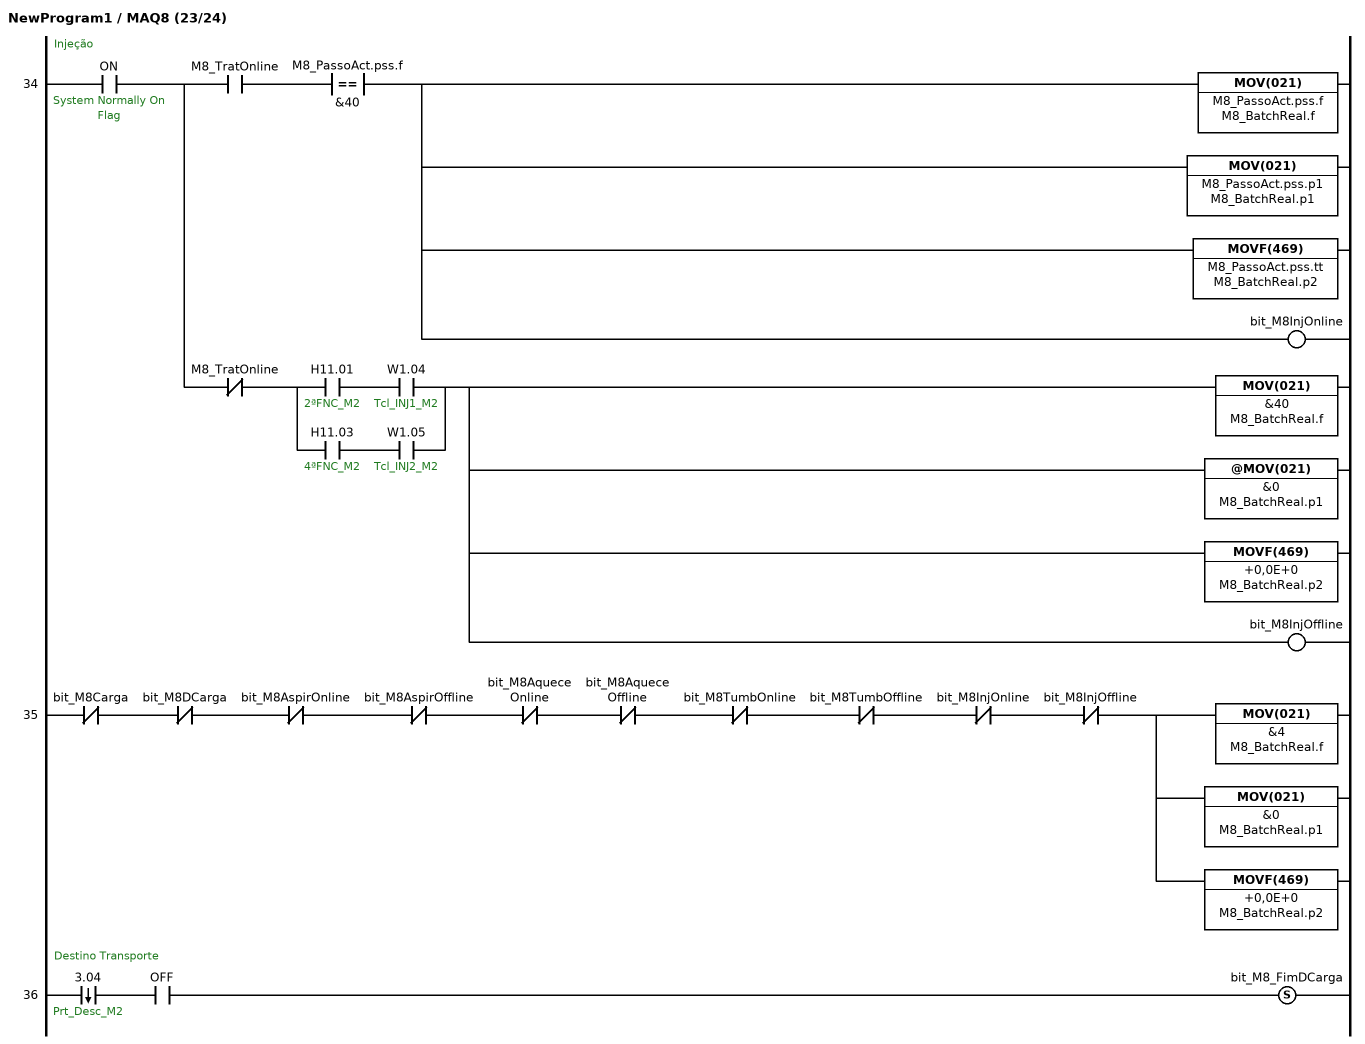
; [picture p48: NewProgram1 / MAQ8, rungs 34-36]
; rung 34: Injeção
LD ON  ; System Normally On Flag
OUT TR0
AND M8_TratOnline
AND=(300) M8_PassoAct.pss.f &40
MOV(021) M8_PassoAct.pss.f M8_BatchReal.f
MOV(021) M8_PassoAct.pss.p1 M8_BatchReal.p1
MOVF(469) M8_PassoAct.pss.tt M8_BatchReal.p2
OUT bit_M8InjOnline
LD TR0
ANDNOT M8_TratOnline
LD H11.01  ; 2ªFNC_M2
AND W1.04  ; Tcl_INJ1_M2
LD H11.03  ; 4ªFNC_M2
AND W1.05  ; Tcl_INJ2_M2
ORLD
ANDLD
MOV(021) &40 M8_BatchReal.f
@MOV(021) &0 M8_BatchReal.p1
MOVF(469) +0,0E+0 M8_BatchReal.p2
OUT bit_M8InjOffline
; rung 35
LDNOT bit_M8Carga
ANDNOT bit_M8DCarga
ANDNOT bit_M8AspirOnline
ANDNOT bit_M8AspirOffline
ANDNOT bit_M8AqueceOnline
ANDNOT bit_M8AqueceOffline
ANDNOT bit_M8TumbOnline
ANDNOT bit_M8TumbOffline
ANDNOT bit_M8InjOnline
ANDNOT bit_M8InjOffline
MOV(021) &4 M8_BatchReal.f
MOV(021) &0 M8_BatchReal.p1
MOVF(469) +0,0E+0 M8_BatchReal.p2
; rung 36: Destino Transporte
%LD 3.04  ; Prt_Desc_M2
AND OFF
SET bit_M8_FimDCarga

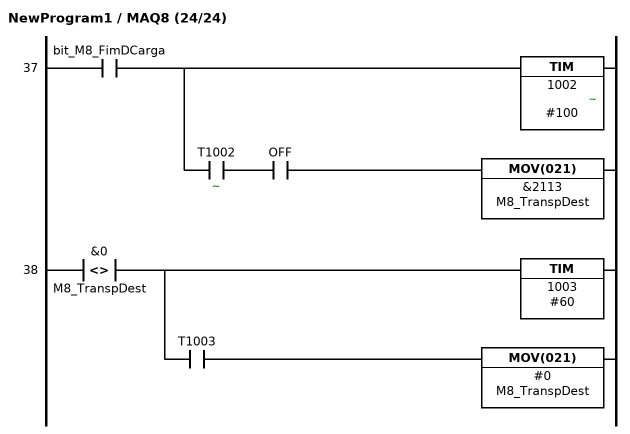
; rung 37
LD bit_M8_FimDCarga
TIM 1002 #100  ; ~
AND T1002  ; ~
AND OFF
MOV(021) &2113 M8_TranspDest
; rung 38
LD<>(305) &0 M8_TranspDest
TIM 1003 #60
AND T1003
MOV(021) #0 M8_TranspDest

### Section TAPETES

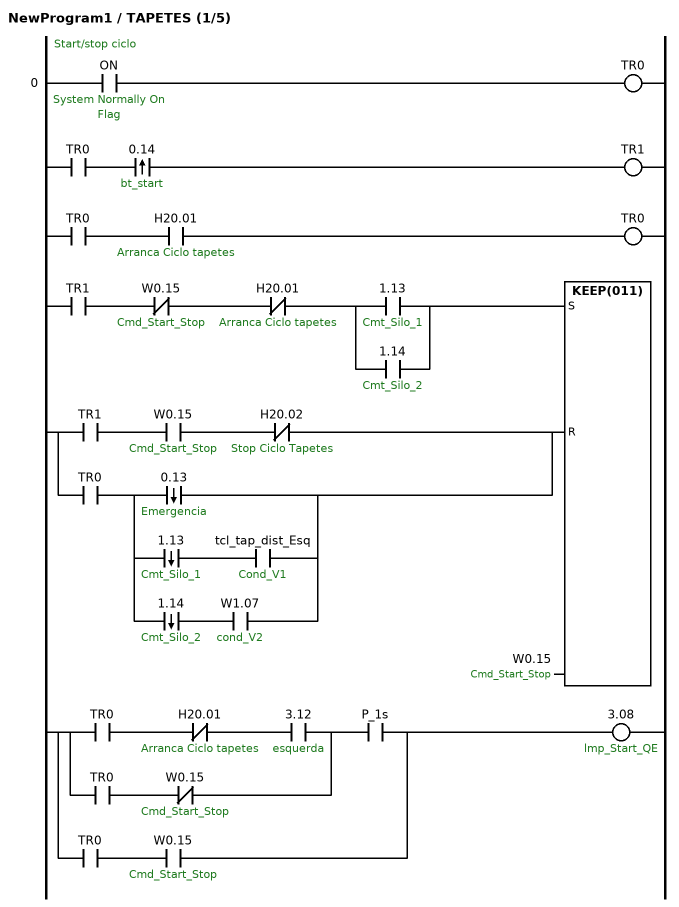
; rung 0: Start/stop ciclo
LD ON  ; System Normally On Flag
OUT TR0
@AND 0.14  ; bt_start
OUT TR1
ANDNOT W0.15  ; Cmd_Start_Stop
ANDNOT H20.01  ; Arranca Ciclo tapetes
LD 1.13  ; Cmt_Silo_1
OR 1.14  ; Cmt_Silo_2
ANDLD
LD TR1
AND W0.15  ; Cmd_Start_Stop
ANDNOT H20.02  ; Stop Ciclo Tapetes
LD TR0
%LD 0.13  ; Emergencia
%LD 1.13  ; Cmt_Silo_1
AND tcl_tap_dist_Esq  ; Cond_V1
ORLD
%LD 1.14  ; Cmt_Silo_2
AND W1.07  ; cond_V2
ORLD
ANDLD
ORLD
KEEP(011) W0.15  ; Cmd_Start_Stop
LD TR0
ANDNOT H20.01  ; Arranca Ciclo tapetes
AND 3.12  ; esquerda
LD TR0
AND H20.01  ; Arranca Ciclo tapetes
OUT TR0
ANDNOT W0.15  ; Cmd_Start_Stop
ORLD
AND P_1s
LD TR0
AND W0.15  ; Cmd_Start_Stop
ORLD
OUT 3.08  ; lmp_Start_QE

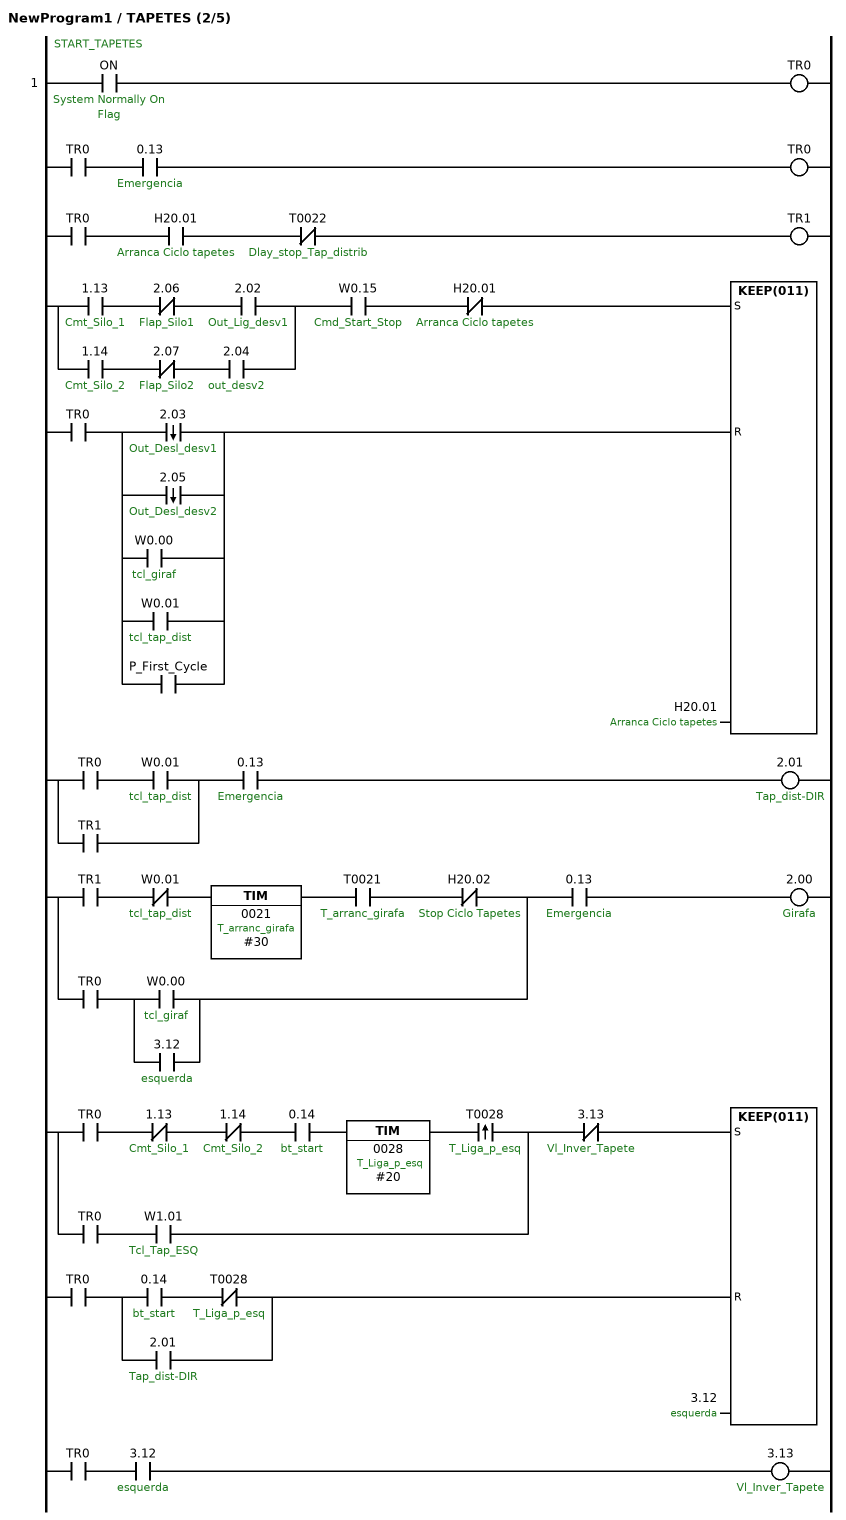
; rung 1: START_TAPETES
LD 1.13  ; Cmt_Silo_1
ANDNOT 2.06  ; Flap_Silo1
AND 2.02  ; Out_Lig_desv1
LD 1.14  ; Cmt_Silo_2
ANDNOT 2.07  ; Flap_Silo2
AND 2.04  ; out_desv2
ORLD
AND W0.15  ; Cmd_Start_Stop
ANDNOT H20.01  ; Arranca Ciclo tapetes
LD ON  ; System Normally On Flag
OUT TR0
%LD 2.03  ; Out_Desl_desv1
%OR 2.05  ; Out_Desl_desv2
OR W0.00  ; tcl_giraf
OR W0.01  ; tcl_tap_dist
OR P_First_Cycle
ANDLD
KEEP(011) H20.01  ; Arranca Ciclo tapetes
LD TR0
AND 0.13  ; Emergencia
OUT TR0
AND W0.01  ; tcl_tap_dist
LD TR0
AND H20.01  ; Arranca Ciclo tapetes
ANDNOT T0022  ; Dlay_stop_Tap_distrib
OUT TR1
ORLD
AND 0.13  ; Emergencia
OUT 2.01  ; Tap_dist-DIR
LD TR1
ANDNOT W0.01  ; tcl_tap_dist
TIM 0021 #30  ; T_arranc_girafa
AND T0021  ; T_arranc_girafa
ANDNOT H20.02  ; Stop Ciclo Tapetes
LD TR0
LD W0.00  ; tcl_giraf
OR 3.12  ; esquerda
ANDLD
ORLD
AND 0.13  ; Emergencia
OUT 2.00  ; Girafa
LD TR0
ANDNOT 1.13  ; Cmt_Silo_1
ANDNOT 1.14  ; Cmt_Silo_2
AND 0.14  ; bt_start
TIM 0028 #20  ; T_Liga_p_esq
@AND T0028  ; T_Liga_p_esq
LD TR0
AND W1.01  ; Tcl_Tap_ESQ
ORLD
ANDNOT 3.13  ; Vl_Inver_Tapete
LD TR0
LD 0.14  ; bt_start
ANDNOT T0028  ; T_Liga_p_esq
OR 2.01  ; Tap_dist-DIR
ANDLD
KEEP(011) 3.12  ; esquerda
LD TR0
AND 3.12  ; esquerda
OUT 3.13  ; Vl_Inver_Tapete

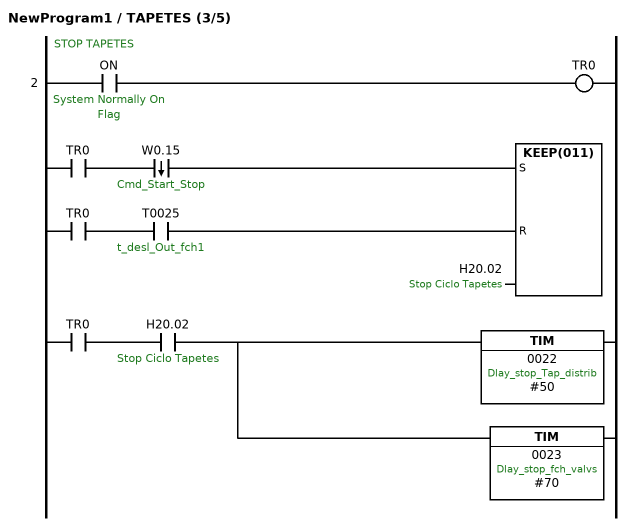
; rung 2: STOP TAPETES
LD ON  ; System Normally On Flag
OUT TR0
%AND W0.15  ; Cmd_Start_Stop
LD TR0
AND T0025  ; t_desl_Out_fch1
KEEP(011) H20.02  ; Stop Ciclo Tapetes
LD TR0
AND H20.02  ; Stop Ciclo Tapetes
TIM 0022 #50  ; Dlay_stop_Tap_distrib
TIM 0023 #70  ; Dlay_stop_fch_valvs

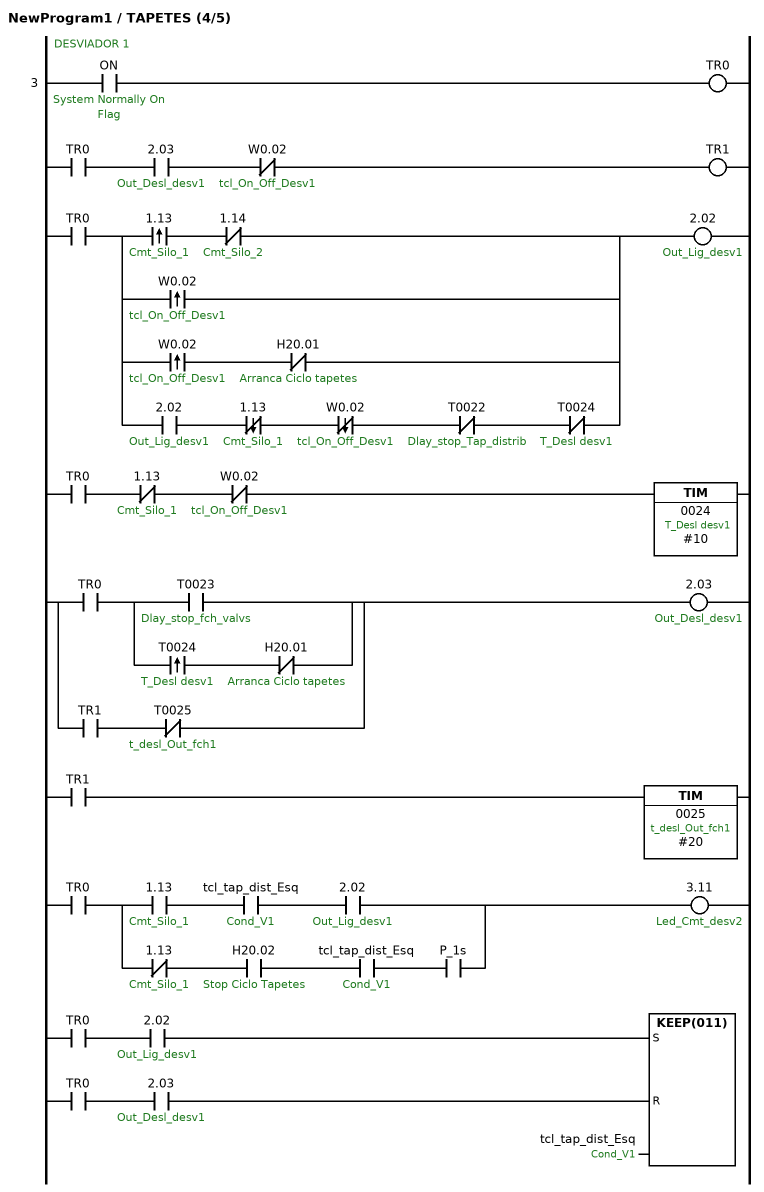
; rung 3: DESVIADOR 1
LD ON  ; System Normally On Flag
OUT TR0
@LD 1.13  ; Cmt_Silo_1
ANDNOT 1.14  ; Cmt_Silo_2
@OR W0.02  ; tcl_On_Off_Desv1
@LD W0.02  ; tcl_On_Off_Desv1
ANDNOT H20.01  ; Arranca Ciclo tapetes
ORLD
LD 2.02  ; Out_Lig_desv1
%ANDNOT 1.13  ; Cmt_Silo_1
%ANDNOT W0.02  ; tcl_On_Off_Desv1
ANDNOT T0022  ; Dlay_stop_Tap_distrib
ANDNOT T0024  ; T_Desl desv1
ORLD
ANDLD
OUT 2.02  ; Out_Lig_desv1
LD TR0
ANDNOT 1.13  ; Cmt_Silo_1
ANDNOT W0.02  ; tcl_On_Off_Desv1
TIM 0024 #10  ; T_Desl desv1
LD TR0
LD T0023  ; Dlay_stop_fch_valvs
@LD T0024  ; T_Desl desv1
ANDNOT H20.01  ; Arranca Ciclo tapetes
ORLD
ANDLD
LD TR0
AND 2.03  ; Out_Desl_desv1
ANDNOT W0.02  ; tcl_On_Off_Desv1
OUT TR1
ANDNOT T0025  ; t_desl_Out_fch1
ORLD
OUT 2.03  ; Out_Desl_desv1
LD TR1
TIM 0025 #20  ; t_desl_Out_fch1
LD TR0
LD 1.13  ; Cmt_Silo_1
AND tcl_tap_dist_Esq  ; Cond_V1
AND 2.02  ; Out_Lig_desv1
LDNOT 1.13  ; Cmt_Silo_1
AND H20.02  ; Stop Ciclo Tapetes
AND tcl_tap_dist_Esq  ; Cond_V1
AND P_1s
ORLD
ANDLD
OUT 3.11  ; Led_Cmt_desv2
LD TR0
AND 2.02  ; Out_Lig_desv1
LD TR0
AND 2.03  ; Out_Desl_desv1
KEEP(011) tcl_tap_dist_Esq  ; Cond_V1

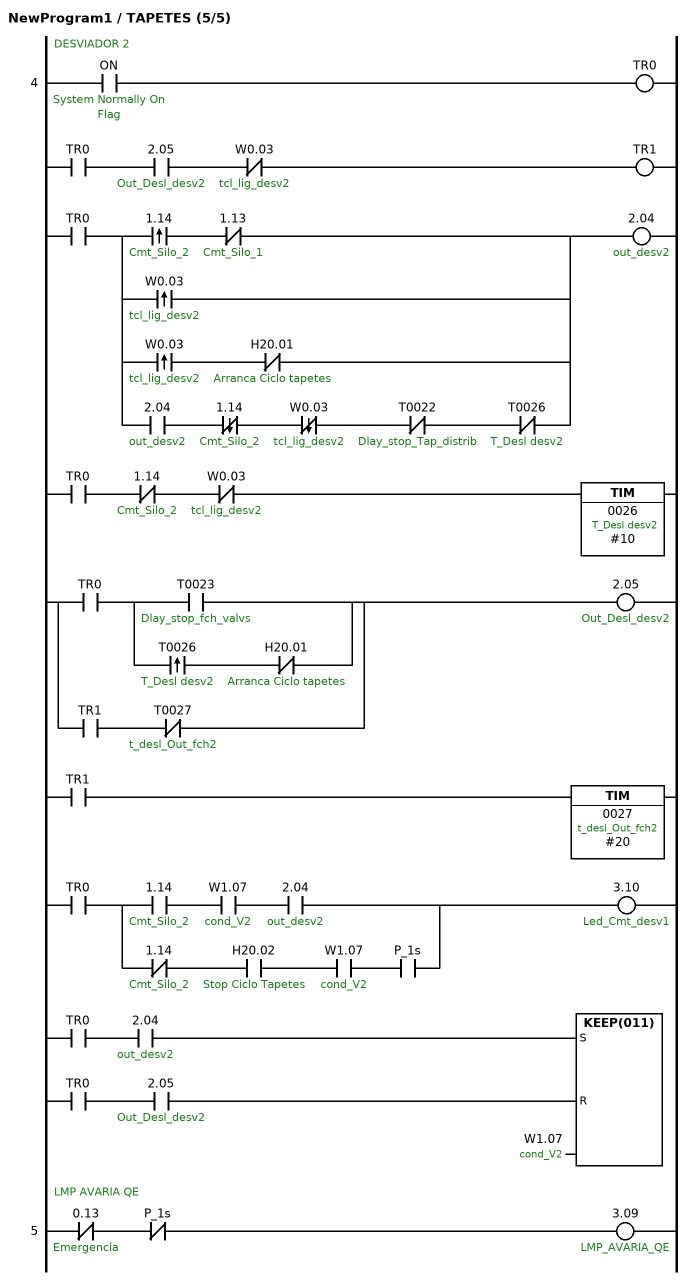
; rung 4: DESVIADOR 2
LD ON  ; System Normally On Flag
OUT TR0
@LD 1.14  ; Cmt_Silo_2
ANDNOT 1.13  ; Cmt_Silo_1
@OR W0.03  ; tcl_lig_desv2
@LD W0.03  ; tcl_lig_desv2
ANDNOT H20.01  ; Arranca Ciclo tapetes
ORLD
LD 2.04  ; out_desv2
%ANDNOT 1.14  ; Cmt_Silo_2
%ANDNOT W0.03  ; tcl_lig_desv2
ANDNOT T0022  ; Dlay_stop_Tap_distrib
ANDNOT T0026  ; T_Desl desv2
ORLD
ANDLD
OUT 2.04  ; out_desv2
LD TR0
ANDNOT 1.14  ; Cmt_Silo_2
ANDNOT W0.03  ; tcl_lig_desv2
TIM 0026 #10  ; T_Desl desv2
LD TR0
LD T0023  ; Dlay_stop_fch_valvs
@LD T0026  ; T_Desl desv2
ANDNOT H20.01  ; Arranca Ciclo tapetes
ORLD
ANDLD
LD TR0
AND 2.05  ; Out_Desl_desv2
ANDNOT W0.03  ; tcl_lig_desv2
OUT TR1
ANDNOT T0027  ; t_desl_Out_fch2
ORLD
OUT 2.05  ; Out_Desl_desv2
LD TR1
TIM 0027 #20  ; t_desl_Out_fch2
LD TR0
LD 1.14  ; Cmt_Silo_2
AND W1.07  ; cond_V2
AND 2.04  ; out_desv2
LDNOT 1.14  ; Cmt_Silo_2
AND H20.02  ; Stop Ciclo Tapetes
AND W1.07  ; cond_V2
AND P_1s
ORLD
ANDLD
OUT 3.10  ; Led_Cmt_desv1
LD TR0
AND 2.04  ; out_desv2
LD TR0
AND 2.05  ; Out_Desl_desv2
KEEP(011) W1.07  ; cond_V2
; rung 5: LMP AVARIA QE
LDNOT 0.13  ; Emergencia
ANDNOT P_1s
OUT 3.09  ; LMP_AVARIA_QE

### Section Comm_Master2Line

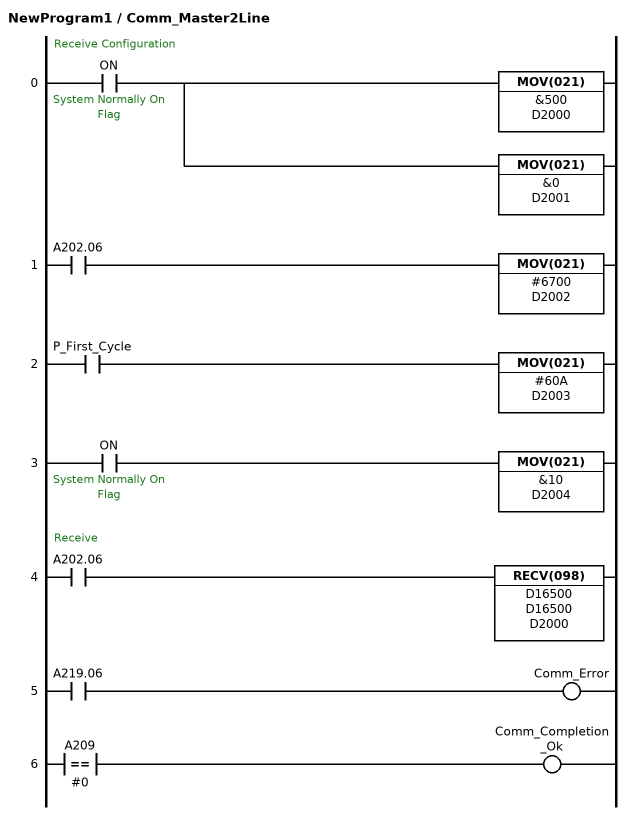
; rung 0: Receive Configuration
LD ON  ; System Normally On Flag
MOV(021) &500 D2000  // Number of the words to read
MOV(021) &0 D2001  // Network Address
; rung 1
LD A202.06
MOV(021) #6700 D2002  // Source's node adress, and unit adress
; rung 2
LD P_First_Cycle
MOV(021) #60A D2003  // ReceiveResponse Required, Logical Port, always 0, and Retries
; rung 3
LD ON  ; System Normally On Flag
MOV(021) &10 D2004  // Timeout
; rung 4: Receive
LD A202.06
RECV(098) D16500 D16500 D2000
; rung 5
LD A219.06
OUT Comm_Error
; rung 6
LD=(300) A209 #0
OUT Comm_Completion_Ok

### Section END
; rung 0
END(001)

## Function block _CPU011_ReceiveData (Omron library block, body left out)

## Function block fb_CopySteps
VAR_INPUT
  Rcp_Ok : BOOL;
END_VAR
VAR_OUTPUT
  Receita_Ok : BOOL;
END_VAR
VAR_IN_OUT
  Recipe : s_of;
  Steps : s_of_net;
END_VAR
Recipe.pss[0].f:=Steps.pss[0].f;
Recipe.pss[0].p1:=Steps.pss[0].p1;
Recipe.pss[0].p2:=Steps.pss[0].p2;
Recipe.pss[0].uni:=0;
Recipe.pss[0].uni:=12;
CASE Recipe.pss[0].f OF
	40:Recipe.pss[0].uni:=9;
END_CASE;

Recipe.pss[1].f:=Steps.pss[1].f;
Recipe.pss[1].p1:=Steps.pss[1].p1;
Recipe.pss[1].p2:=Steps.pss[1].p2;
Recipe.pss[1].uni:=0;
Recipe.pss[1].uni:=12;
CASE Recipe.pss[1].f OF
	40:Recipe.pss[1].uni:=9;
END_CASE;

Recipe.pss[2].f:=Steps.pss[2].f;
Recipe.pss[2].p1:=Steps.pss[2].p1;
Recipe.pss[2].p2:=Steps.pss[2].p2;
Recipe.pss[2].uni:=0;
Recipe.pss[2].uni:=12;
CASE Recipe.pss[2].f OF
	40:Recipe.pss[2].uni:=9;
END_CASE;

Recipe.pss[3].f:=Steps.pss[3].f;
Recipe.pss[3].p1:=Steps.pss[3].p1;
Recipe.pss[3].p2:=Steps.pss[3].p2;
Recipe.pss[3].uni:=0;
Recipe.pss[3].uni:=12;
CASE Recipe.pss[3].f OF
	40:Recipe.pss[3].uni:=9;
END_CASE;

Recipe.pss[4].f:=Steps.pss[4].f;
Recipe.pss[4].p1:=Steps.pss[4].p1;
Recipe.pss[4].p2:=Steps.pss[4].p2;
Recipe.pss[4].uni:=0;
Recipe.pss[4].uni:=12;
CASE Recipe.pss[4].f OF
	40:Recipe.pss[4].uni:=9;
END_CASE;

Recipe.pss[5].f:=Steps.pss[5].f;
Recipe.pss[5].p1:=Steps.pss[5].p1;
Recipe.pss[5].p2:=Steps.pss[5].p2;
Recipe.pss[5].uni:=0;
Recipe.pss[5].uni:=12;
CASE Recipe.pss[5].f OF
	40:Recipe.pss[5].uni:=9;
END_CASE;

Recipe.pss[6].f:=Steps.pss[6].f;
Recipe.pss[6].p1:=Steps.pss[6].p1;
Recipe.pss[6].p2:=Steps.pss[6].p2;
Recipe.pss[6].uni:=0;
Recipe.pss[6].uni:=12;
CASE Recipe.pss[6].f OF
	40:Recipe.pss[6].uni:=9;
END_CASE;

Recipe.pss[7].f:=Steps.pss[7].f;
Recipe.pss[7].p1:=Steps.pss[7].p1;
Recipe.pss[7].p2:=Steps.pss[7].p2;
Recipe.pss[7].uni:=0;
Recipe.pss[7].uni:=12;
CASE Recipe.pss[7].f OF
	40:Recipe.pss[7].uni:=9;
END_CASE;

Recipe.pss[8].f:=Steps.pss[8].f;
Recipe.pss[8].p1:=Steps.pss[8].p1;
Recipe.pss[8].p2:=Steps.pss[8].p2;
Recipe.pss[8].uni:=0;
Recipe.pss[8].uni:=12;
CASE Recipe.pss[8].f OF
	40:Recipe.pss[8].uni:=9;
END_CASE;

Recipe.pss[9].f:=Steps.pss[9].f;
Recipe.pss[9].p1:=Steps.pss[9].p1;
Recipe.pss[9].p2:=Steps.pss[9].p2;
Recipe.pss[9].uni:=0;
Recipe.pss[9].uni:=12;
CASE Recipe.pss[9].f OF
	40:Recipe.pss[9].uni:=9;
END_CASE;

Recipe.pss[10].f:=Steps.pss[10].f;
Recipe.pss[10].p1:=Steps.pss[10].p1;
Recipe.pss[10].p2:=Steps.pss[10].p2;
Recipe.pss[10].uni:=0;
Recipe.pss[10].uni:=12;
CASE Recipe.pss[10].f OF
	40:Recipe.pss[10].uni:=9;
END_CASE;

Recipe.pss[11].f:=Steps.pss[11].f;
Recipe.pss[11].p1:=Steps.pss[11].p1;
Recipe.pss[11].p2:=Steps.pss[11].p2;
Recipe.pss[11].uni:=0;
Recipe.pss[11].uni:=12;
CASE Recipe.pss[11].f OF
	40:Recipe.pss[11].uni:=9;
END_CASE;
	
Receita_Ok:= Rcp_Ok;

## Function block fb_maquina_mov_pss_act
; FUNÇÃO MAQUINA MOVE PASSOS ACTUAIS - Faz a passagem da função do passo actual da maquina para a zona de memoria do passo actual. Faz também a passagem do total do passo em execução.
VAR_IN_OUT
  passo_act : s_pss_exe;  (* Passo atual em execução *)
  of_exe : s_of;  (* Ordem de fabrico *)
END_VAR
(*Não esta a executar nenhum passo - Limpeza da zona de memória do passo actual*)
	IF (passo_act.num_pss=-1) THEN
		passo_act.pss.f:= 0;
		passo_act.pss.p1:= 0;
		passo_act.pss.p2:=0,0;
		passo_act.pss.tt:= 0,0;
		passo_act.pss.uni:= 0;
	END_IF;
	IF passo_act.num_pss=0 THEN
		passo_act.pss.f:= of_exe.pss[0].f;
		passo_act.pss.p1:= of_exe.pss[0].p1;
		passo_act.pss.p2:= of_exe.pss[0].p2;
		of_exe.pss[0].tt:= passo_act.pss.tt;
		passo_act.pss.uni:=of_exe.pss[0].uni;
	END_IF;
	
		CASE passo_act.num_pss OF
			0: 
				passo_act.pss.f:= of_exe.pss[0].f;
				passo_act.pss.p1:= of_exe.pss[0].p1;
				passo_act.pss.p2:= of_exe.pss[0].p2;
				of_exe.pss[0].tt:= passo_act.pss.tt;
				passo_act.pss.uni:=of_exe.pss[0].uni;
			1: 
				passo_act.pss.f:= of_exe.pss[1].f;
				passo_act.pss.p1:= of_exe.pss[1].p1;
				passo_act.pss.p2:= of_exe.pss[1].p2;
				of_exe.pss[1].tt:= passo_act.pss.tt;
				passo_act.pss.uni:=of_exe.pss[1].uni;
			2:
				passo_act.pss.f:= of_exe.pss[2].f;
				passo_act.pss.p1:= of_exe.pss[2].p1;
				passo_act.pss.p2:= of_exe.pss[2].p2;
				of_exe.pss[2].tt:= passo_act.pss.tt;
				passo_act.pss.uni:=of_exe.pss[2].uni;
			3:
				passo_act.pss.f:= of_exe.pss[3].f;
				passo_act.pss.p1:= of_exe.pss[3].p1;
				passo_act.pss.p2:= of_exe.pss[3].p2;
				of_exe.pss[3].tt:= passo_act.pss.tt;
				passo_act.pss.uni:=of_exe.pss[3].uni;
			4:
				passo_act.pss.f:= of_exe.pss[4].f;
				passo_act.pss.p1:= of_exe.pss[4].p1;
				passo_act.pss.p2:= of_exe.pss[4].p2;
				of_exe.pss[4].tt:= passo_act.pss.tt;
				passo_act.pss.uni:=of_exe.pss[4].uni;
			5:
				passo_act.pss.f:= of_exe.pss[5].f;
				passo_act.pss.p1:= of_exe.pss[5].p1;
				passo_act.pss.p2:= of_exe.pss[5].p2;
				of_exe.pss[5].tt:= passo_act.pss.tt;
				passo_act.pss.uni:=of_exe.pss[5].uni;
			6:
				passo_act.pss.f:= of_exe.pss[6].f;
				passo_act.pss.p1:= of_exe.pss[6].p1;
				passo_act.pss.p2:= of_exe.pss[6].p2;
				of_exe.pss[6].tt:= passo_act.pss.tt;
				passo_act.pss.uni:=of_exe.pss[6].uni;
			7:
				passo_act.pss.f:= of_exe.pss[7].f;
				passo_act.pss.p1:= of_exe.pss[7].p1;
				passo_act.pss.p2:= of_exe.pss[7].p2;
				of_exe.pss[7].tt:= passo_act.pss.tt;
				passo_act.pss.uni:=of_exe.pss[7].uni;
			8:
				passo_act.pss.f:= of_exe.pss[8].f;
				passo_act.pss.p1:= of_exe.pss[8].p1;
				passo_act.pss.p2:= of_exe.pss[8].p2;
				of_exe.pss[8].tt:= passo_act.pss.tt;
				passo_act.pss.uni:=of_exe.pss[8].uni;
			9:
				passo_act.pss.f:= of_exe.pss[9].f;
				passo_act.pss.p1:= of_exe.pss[9].p1;
				passo_act.pss.p2:= of_exe.pss[9].p2;
				of_exe.pss[9].tt:= passo_act.pss.tt;
				passo_act.pss.uni:=of_exe.pss[9].uni;
			10:
				passo_act.pss.f:= of_exe.pss[10].f;
				passo_act.pss.p1:= of_exe.pss[10].p1;
				passo_act.pss.p2:= of_exe.pss[10].p2;
				of_exe.pss[10].tt:= passo_act.pss.tt;
				passo_act.pss.uni:=of_exe.pss[10].uni;
			11:
				passo_act.pss.f:= of_exe.pss[11].f;
				passo_act.pss.p1:= of_exe.pss[11].p1;
				passo_act.pss.p2:= of_exe.pss[11].p2;
				of_exe.pss[11].tt:= passo_act.pss.tt;
				passo_act.pss.uni:=of_exe.pss[11].uni;
		END_CASE;

## Function block fb_maquina_pss_2_str10_PT
; FUNÇÃO PASSO PARA STRING - Transforma os passo em execução em strings para apresentar no HMI.
VAR_IN_OUT
  receita : s_of;  (* Programa *)
  str_pss0 : STRING;  (* String do passo *)
  str_pss1 : STRING;  (* String do passo *)
  str_pss2 : STRING;  (* String do passo *)
  str_pss3 : STRING;  (* String do passo *)
  str_pss4 : STRING;  (* String do passo *)
  str_pss5 : STRING;  (* String do passo *)
  str_pss6 : STRING;  (* String do passo *)
  str_pss7 : STRING;  (* String do passo *)
  str_pss8 : STRING;  (* String do passo *)
  str_pss9 : STRING;  (* String do passo *)
  str_pss10 : STRING;
  str_pss11 : STRING;
  str_act : STRING;  (* String do passo actual *)
  ProgrAct : s_pss_exe;  (* Passo em execução *)
END_VAR
VAR
  str_p1 : STRING;  (* Parametro 1 *)
  str_p2 : STRING;  (* Parametro 2 *)
  dd : REAL;  (* Dividendo *)
  dv : REAL;  (* Divisor *)
  qc : REAL;  (* Quociente *)
  r : REAL;  (* Resto *)
  i : INT;
  pss : s_of_pss;  (* Passo *)
  str_pss : STRING;  (* String do passo *)
END_VAR
FOR i:= 0 TO 11 DO
	(*Passagem dos dados dos varios passos*)
	CASE i OF
		0:
			pss.f:= receita.pss[0].f;
			pss.p1:= receita.pss[0].p1;
			pss.p2:=receita.pss[0].p2;
		1:
			pss.f:= receita.pss[1].f;
			pss.p1:= receita.pss[1].p1;
			pss.p2:=receita.pss[1].p2;
		2:
			pss.f:= receita.pss[2].f;
			pss.p1:= receita.pss[2].p1;
			pss.p2:=receita.pss[2].p2;
		3:
			pss.f:= receita.pss[3].f;
			pss.p1:= receita.pss[3].p1;
			pss.p2:=receita.pss[3].p2;
		4:
			pss.f:= receita.pss[4].f;
			pss.p1:= receita.pss[4].p1;
			pss.p2:=receita.pss[4].p2;
		5:
			pss.f:= receita.pss[5].f;
			pss.p1:= receita.pss[5].p1;
			pss.p2:=receita.pss[5].p2;
		6:
			pss.f:= receita.pss[6].f;
			pss.p1:= receita.pss[6].p1;
			pss.p2:=receita.pss[6].p2;
		7:
			pss.f:= receita.pss[7].f;
			pss.p1:= receita.pss[7].p1;
			pss.p2:=receita.pss[7].p2;
		8:
			pss.f:= receita.pss[8].f;
			pss.p1:= receita.pss[8].p1;
			pss.p2:=receita.pss[8].p2;
		9:
			pss.f:= receita.pss[9].f;
			pss.p1:= receita.pss[9].p1;
			pss.p2:=receita.pss[9].p2;
		10:
			pss.f:= receita.pss[10].f;
			pss.p1:= receita.pss[10].p1;
			pss.p2:=receita.pss[10].p2;
		11:
			pss.f:= receita.pss[11].f;
			pss.p1:= receita.pss[11].p1;
			pss.p2:=receita.pss[11].p2;
		
	END_CASE;
	
	(*Inicialização*)
		str_pss:= '';
 
 	(*Transformação dos valores em string*)
	 str_p1:= INT_TO_STRING(pss.p1);
 
 	dd:= pss.p2*10,0;
 	dv:= 10,0;
 	qc:=INT_TO_REAL(REAL_TO_INT(dd/dv));
 	r:= dd-dv*qc;
	IF r<0,0 THEN
		qc:= qc-1,0;
		r:= 10,0+r;
	END_IF;
	
 	str_p2:= CONCAT(INT_TO_STRING(REAL_TO_INT(qc)),',',INT_TO_STRING(REAL_TO_INT(r)));

  	(*Aspiração*)
 	IF pss.f=10 THEN
		 str_pss:=CONCAT('Aspirazione ',str_p1,'s');
	END_IF;

	(*Aquecimento*)
 	IF pss.f=20 THEN
		 str_pss:=CONCAT('Riscaldamento ',str_p2,'ºC ',str_p1,'s');
	END_IF;

  	(*Tratamento*)
 	IF pss.f=30 THEN
		 str_pss:=CONCAT('Trattamento ',str_p1,'s');
	END_IF;

  	(*Injecção*)
 	IF pss.f=40 THEN
		 CASE pss.p1 OF
		 	1:str_pss:=CONCAT('BOPSIL ',str_p2,'ml');  (*BOPSIL*)
			2:str_pss:=CONCAT('P28 ',str_p2,'ml');  (*P28*)
			3:str_pss:=CONCAT('SILBIONE ',str_p2,'ml');  (*SILICONE*)
			4:str_pss:=CONCAT('P2X ',str_p2,'ml');  (*P2X*)
			5:str_pss:=CONCAT('LC104 ',str_p2,'ml');  (*LC104*)
			6:str_pss:=CONCAT('PARAFFINA ',str_p2,'ml');  (*PARAFINA*)
			7:str_pss:=CONCAT('TEFLON ',str_p2,'ml');  (*TEFLON*)
			8:str_pss:=CONCAT('CAF ',str_p2,'ml');  (*CAF*)
			9:str_pss:=CONCAT('X15 ',str_p2,'ml');  (*X15*)
			10:str_pss:=CONCAT('SWAM P.N.S. ',str_p2,'ml');  (*SWAM P.N.S.*)
			11:str_pss:=CONCAT('SWAM P.SA ',str_p2,'ml');  (*SWAM P.SA*)		
			19:str_pss:=CONCAT('TR02 ',str_p2,'ml');  (*TR02*)
		END_CASE;
	END_IF;

  	(*LOAD*)
 	IF pss.f=70 THEN
		 str_pss:='Carico ';
	END_IF;

  	(*UNLOAD*)
 	IF pss.f=80 THEN
		 str_pss:='Scarico ';
	END_IF;
	
	(*Passagem das strings dos varios passos*)
	CASE i OF
		0:	str_pss0:= str_pss;
		1:	str_pss1:= str_pss;
		2:	str_pss2:= str_pss;
		3:	str_pss3:= str_pss;
		4:	str_pss4:= str_pss;
		5:	str_pss5:= str_pss;
		6:	str_pss6:= str_pss;
		7:	str_pss7:= str_pss;
		8:	str_pss8:= str_pss;
		9:	str_pss9:= str_pss;
		10:	str_pss10:= str_pss;
		11:	str_pss11:= str_pss;
	END_CASE;
	
	(*String do passo actual*)
	str_act:= '';
	CASE ProgrAct.num_pss OF
		0:	str_act:= str_pss0;
		1:	str_act:= str_pss1;
		2:	str_act:= str_pss2;
		3:	str_act:= str_pss3;
		4:	str_act:= str_pss4;
		5:	str_act:= str_pss5;
		6:	str_act:= str_pss6;
		7:	str_act:= str_pss7;
		8:	str_act:= str_pss8;
		9:	str_act:= str_pss9;
		10:	str_act:= str_pss10;
		11:	str_act:= str_pss11;
	END_CASE;
		
END_FOR;

## Function block fb_of_clear
; FUNÇÃO LIMPA UMA ORDEM DE FABRICO - Coloca os valores da OF a zero.
VAR_INPUT
  Start : BOOL;
END_VAR
VAR_OUTPUT
  End : BOOL;
END_VAR
VAR_IN_OUT
  of_in_out : s_of;  (* OF a ser apagada *)
END_VAR
IF (Start=TRUE AND End=FALSE) THEN
	of_in_out.pss[0].f:= 0;
	of_in_out.pss[0].p1:=0;
	of_in_out.pss[0].p2:=0,0;
	of_in_out.pss[0].tt:=0,0;
	of_in_out.pss[0].uni:=0;
	of_in_out.pss[0].uni:=12;
	CASE of_in_out.pss[0].f OF
		40:of_in_out.pss[0].uni:=9;
	END_CASE;
	
	of_in_out.pss[1].f:= 0;
	of_in_out.pss[1].p1:=0;
	of_in_out.pss[1].p2:=0,0;
	of_in_out.pss[1].tt:=0,0;
	of_in_out.pss[1].uni:=1;
	of_in_out.pss[1].uni:=12;
	CASE of_in_out.pss[1].f OF
		40:of_in_out.pss[1].uni:=9;
	END_CASE;
	
	of_in_out.pss[2].f:= 0;
	of_in_out.pss[2].p1:=0;
	of_in_out.pss[2].p2:=0,0;
	of_in_out.pss[2].tt:=0,0;
	of_in_out.pss[2].uni:=1;
	of_in_out.pss[2].uni:=12;
	CASE of_in_out.pss[2].f OF
		40:of_in_out.pss[2].uni:=9;
	END_CASE;
	
	of_in_out.pss[3].f:= 0;
	of_in_out.pss[3].p1:=0;
	of_in_out.pss[3].p2:=0,0;
	of_in_out.pss[3].tt:=0,0;
	of_in_out.pss[3].uni:=1;
	of_in_out.pss[3].uni:=12;
	CASE of_in_out.pss[3].f OF
		40:of_in_out.pss[3].uni:=9;
	END_CASE;
	
	of_in_out.pss[4].f:= 0;
	of_in_out.pss[4].p1:=0;
	of_in_out.pss[4].p2:=0,0;
	of_in_out.pss[4].tt:=0,0;
	of_in_out.pss[4].uni:=1;
	of_in_out.pss[4].uni:=12;
	CASE of_in_out.pss[4].f OF
		40:of_in_out.pss[4].uni:=9;
	END_CASE;
	
	of_in_out.pss[5].f:= 0;
	of_in_out.pss[5].p1:=0;
	of_in_out.pss[5].p2:=0,0;
	of_in_out.pss[5].tt:=0,0;
	of_in_out.pss[5].uni:=1;
	of_in_out.pss[5].uni:=12;
	CASE of_in_out.pss[5].f OF
		40:of_in_out.pss[5].uni:=9;
	END_CASE;
	
	of_in_out.pss[6].f:= 0;
	of_in_out.pss[6].p1:=0;
	of_in_out.pss[6].p2:=0,0;
	of_in_out.pss[6].tt:=0,0;
	of_in_out.pss[6].uni:=1;
	of_in_out.pss[6].uni:=12;
	CASE of_in_out.pss[6].f OF
		40:of_in_out.pss[6].uni:=9;
	END_CASE;
	
	of_in_out.pss[7].f:= 0;
	of_in_out.pss[7].p1:=0;
	of_in_out.pss[7].p2:=0,0;
	of_in_out.pss[7].tt:=0,0;
	of_in_out.pss[7].uni:=1;
	of_in_out.pss[7].uni:=12;
	CASE of_in_out.pss[7].f OF
		40:of_in_out.pss[7].uni:=9;
	END_CASE;
	
	of_in_out.pss[8].f:= 0;
	of_in_out.pss[8].p1:=0;
	of_in_out.pss[8].p2:=0,0;
	of_in_out.pss[8].tt:=0,0;
	of_in_out.pss[8].uni:=1;
	of_in_out.pss[8].uni:=12;
	CASE of_in_out.pss[8].f OF
		40:of_in_out.pss[8].uni:=9;
	END_CASE;
	
	of_in_out.pss[9].f:= 0;
	of_in_out.pss[9].p1:=0;
	of_in_out.pss[9].p2:=0,0;
	of_in_out.pss[9].tt:=0,0;
	of_in_out.pss[9].uni:=1;
	of_in_out.pss[9].uni:=12;
	CASE of_in_out.pss[9].f OF
		40:of_in_out.pss[9].uni:=9;
	END_CASE;
	
	of_in_out.pss[10].f:= 0;
	of_in_out.pss[10].p1:=0;
	of_in_out.pss[10].p2:=0,0;
	of_in_out.pss[10].tt:=0,0;
	of_in_out.pss[10].uni:=1;
	of_in_out.pss[10].uni:=12;
	CASE of_in_out.pss[10].f OF
		40:of_in_out.pss[10].uni:=9;
	END_CASE;
	
	of_in_out.pss[11].f:= 0;
	of_in_out.pss[11].p1:=0;
	of_in_out.pss[11].p2:=0,0;
	of_in_out.pss[11].tt:=0,0;
	of_in_out.pss[11].uni:=1;
	of_in_out.pss[11].uni:=12;
	CASE of_in_out.pss[11].f OF
		40:of_in_out.pss[11].uni:=9;
	END_CASE;
	
	End:= TRUE;
ELSIF Start=FALSE THEN
	End:= FALSE;
END_IF;

## Function block fb_of_copy
; FUNÇÃO COPIA ORDENS DE FABRICO - Copia ordens de fabrico.
VAR_INPUT
  Start : BOOL;
END_VAR
VAR_OUTPUT
  End : BOOL;
END_VAR
VAR_IN_OUT
  of_in : s_of;  (* OF original *)
  of_out : s_of;  (* OF para onde faz a copia *)
END_VAR
IF (Start=TRUE AND End=FALSE) THEN
	of_out.pss[0].f:=of_in.pss[0].f;
	of_out.pss[0].p1:=of_in.pss[0].p1;
	of_out.pss[0].p2:=of_in.pss[0].p2;
	of_out.pss[0].tt:=of_in.pss[0].tt;
	of_out.pss[0].uni:=0;
	of_out.pss[0].uni:=12;
	CASE of_out.pss[0].f OF
		40:of_out.pss[0].uni:=9;
	END_CASE;
	
	of_out.pss[1].f:=of_in.pss[1].f;
	of_out.pss[1].p1:=of_in.pss[1].p1;
	of_out.pss[1].p2:=of_in.pss[1].p2;
	of_out.pss[1].tt:=of_in.pss[1].tt;
	of_out.pss[1].uni:=0;
	of_out.pss[1].uni:=12;
	CASE of_out.pss[1].f OF
		40:of_out.pss[1].uni:=9;
	END_CASE;
		
	of_out.pss[2].f:=of_in.pss[2].f;
	of_out.pss[2].p1:=of_in.pss[2].p1;
	of_out.pss[2].p2:=of_in.pss[2].p2;
	of_out.pss[2].tt:=of_in.pss[2].tt;
	of_out.pss[2].uni:=0;
	of_out.pss[2].uni:=12;
	CASE of_out.pss[2].f OF
		40:of_out.pss[2].uni:=9;
	END_CASE;
	
	of_out.pss[3].f:=of_in.pss[3].f;
	of_out.pss[3].p1:=of_in.pss[3].p1;
	of_out.pss[3].p2:=of_in.pss[3].p2;
	of_out.pss[3].tt:=of_in.pss[3].tt;
	of_out.pss[3].uni:=0;
	of_out.pss[3].uni:=12;
	CASE of_out.pss[3].f OF
		40:of_out.pss[3].uni:=9;
	END_CASE;
	
	of_out.pss[4].f:=of_in.pss[4].f;
	of_out.pss[4].p1:=of_in.pss[4].p1;
	of_out.pss[4].p2:=of_in.pss[4].p2;
	of_out.pss[4].tt:=of_in.pss[4].tt;
	of_out.pss[4].uni:=0;
	of_out.pss[4].uni:=12;
	CASE of_out.pss[4].f OF
		40:of_out.pss[4].uni:=9;
	END_CASE;
	
	of_out.pss[5].f:=of_in.pss[5].f;
	of_out.pss[5].p1:=of_in.pss[5].p1;
	of_out.pss[5].p2:=of_in.pss[5].p2;
	of_out.pss[5].tt:=of_in.pss[5].tt;
	of_out.pss[5].uni:=0;
	of_out.pss[5].uni:=12;
	CASE of_out.pss[5].f OF
		40:of_out.pss[5].uni:=9;
	END_CASE;
	
	of_out.pss[6].f:=of_in.pss[6].f;
	of_out.pss[6].p1:=of_in.pss[6].p1;
	of_out.pss[6].p2:=of_in.pss[6].p2;
	of_out.pss[6].tt:=of_in.pss[6].tt;
	of_out.pss[6].uni:=0;
	of_out.pss[6].uni:=12;
	CASE of_out.pss[6].f OF
		40:of_out.pss[6].uni:=9;
	END_CASE;
	
	of_out.pss[7].f:=of_in.pss[7].f;
	of_out.pss[7].p1:=of_in.pss[7].p1;
	of_out.pss[7].p2:=of_in.pss[7].p2;
	of_out.pss[7].tt:=of_in.pss[7].tt;
	of_out.pss[7].uni:=0;
	of_out.pss[7].uni:=12;
	CASE of_out.pss[7].f OF
		40:of_out.pss[7].uni:=9;
	END_CASE;
	
	of_out.pss[8].f:=of_in.pss[8].f;
	of_out.pss[8].p1:=of_in.pss[8].p1;
	of_out.pss[8].p2:=of_in.pss[8].p2;
	of_out.pss[8].tt:=of_in.pss[8].tt;
	of_out.pss[8].uni:=0;
	of_out.pss[8].uni:=12;
	CASE of_out.pss[8].f OF
		40:of_out.pss[8].uni:=9;
	END_CASE;
	
	of_out.pss[9].f:=of_in.pss[9].f;
	of_out.pss[9].p1:=of_in.pss[9].p1;
	of_out.pss[9].p2:=of_in.pss[9].p2;
	of_out.pss[9].tt:=of_in.pss[9].tt;
	of_out.pss[9].uni:=0;
	of_out.pss[9].uni:=12;
	CASE of_out.pss[9].f OF
		40:of_out.pss[9].uni:=9;
	END_CASE;
	
	of_out.pss[10].f:=of_in.pss[10].f;
	of_out.pss[10].p1:=of_in.pss[10].p1;
	of_out.pss[10].p2:=of_in.pss[10].p2;
	of_out.pss[10].tt:=of_in.pss[10].tt;
	of_out.pss[10].uni:=0;
	of_out.pss[10].uni:=12;
	CASE of_out.pss[10].f OF
		40:of_out.pss[10].uni:=9;
	END_CASE;
	
	of_out.pss[11].f:=of_in.pss[11].f;
	of_out.pss[11].p1:=of_in.pss[11].p1;
	of_out.pss[11].p2:=of_in.pss[11].p2;
	of_out.pss[11].tt:=of_in.pss[11].tt;
	of_out.pss[11].uni:=0;
	of_out.pss[11].uni:=12;
	CASE of_out.pss[11].f OF
		40:of_out.pss[11].uni:=9;
	END_CASE;
	
	End:= TRUE;
ELSIF Start=FALSE THEN	
	End:= FALSE;
END_IF;

## Function block Maquina
VAR_INPUT
  Carga_On : BOOL;  (* Carga ativa *)
  DCarga_On : BOOL;  (* Descarga ativa *)
  Aquece_On : BOOL;  (* Aquecimento ativo *)
  Rotacao_On : BOOL;  (* Rotação ativa *)
  Aspir_On : BOOL;  (* Aspiração ativa *)
  Injecao_Ok : BOOL;  (* Produto Injetado *)
  Avaria : BOOL;
  Start : BOOL;  (* Início Ciclo *)
  Stop : BOOL;
  MqDisponivel : BOOL;
  Offline : BOOL;
END_VAR
VAR_OUTPUT
  Temperatura : INT;
END_VAR
VAR_IN_OUT
  rcpMoe : s_of;  (* Receita Moega *)
  rcpMq : s_of;  (* Receita máquina *)
  stp : s_pss_exe;  (* Passo atual *)
  trat : s_trat;
  Estado : s_Estado;
  rcpMoega_Ok : BOOL;
  rcpMaquina_Ok : BOOL;
  Auto : BOOL;
END_VAR
VAR
  Ctrl : INT;
  moega_to_maq : fb_of_copy;
  bit_MoveRcp : BOOL;
  bit_MoveRcp_End : BOOL;
  rcp_del : fb_of_clear;
  bit_DelRcp_End : BOOL;
  aux_MoveRcp : BOOL;
  mov_step : fb_maquina_mov_pss_act;
  T_Stop : TIMER;
  rcpMq_del : fb_of_clear;
  bit_DelRcpMq_End : BOOL;
  bit_DCargaFim : BOOL;
  aux_Rotacao : BOOL;
  param : REAL;
  memCtrl : INT;
  auxAspira : BOOL;
  T_muda : TIMER;
  T_Stop1 : TIMER;
  tmpTemper : REAL;
  bit_FimInjec : BOOL;
  T_FimInjec : TIMER;
  Estado_delay : TIMER;
  ciclo_holder : BOOL;
  StpHolder : BOOL;
  StpHolder_T : TIMER;
END_VAR

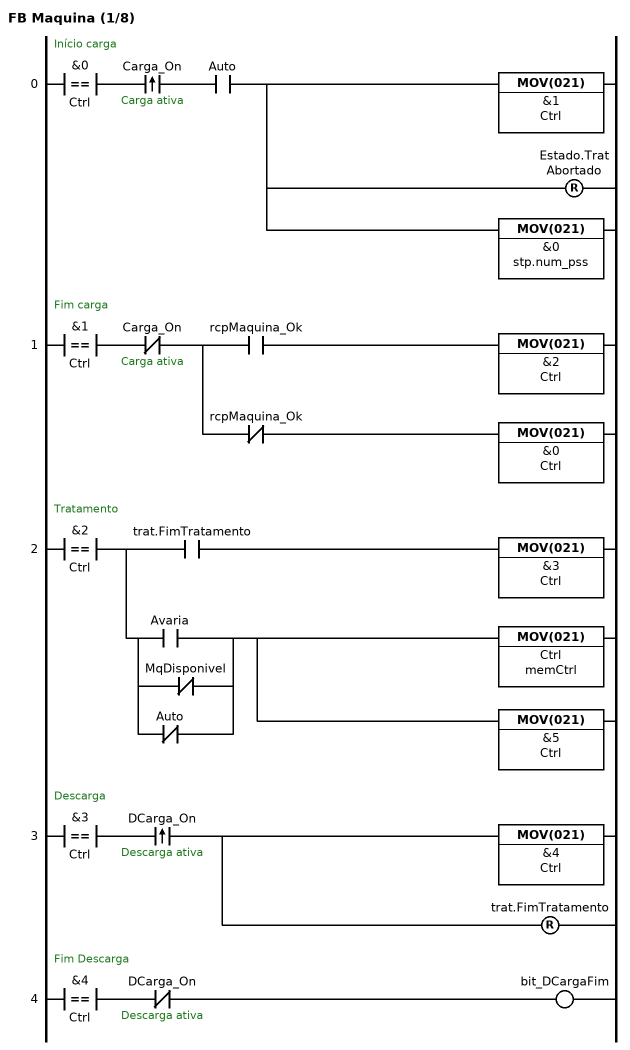
; rung 0: Início carga
LD=(300) &0 Ctrl
@AND Carga_On  ; Carga ativa
AND Auto
MOV(021) &1 Ctrl
RSET Estado.TratAbortado
MOV(021) &0 stp.num_pss
; rung 1: Fim carga
LD=(300) &1 Ctrl
ANDNOT Carga_On  ; Carga ativa
OUT TR0
AND rcpMaquina_Ok
MOV(021) &2 Ctrl
LD TR0
ANDNOT rcpMaquina_Ok
MOV(021) &0 Ctrl
; rung 2: Tratamento
LD=(300) &2 Ctrl
OUT TR0
AND trat.FimTratamento
MOV(021) &3 Ctrl
LD TR0
LD Avaria
ORNOT MqDisponivel
ORNOT Auto
ANDLD
MOV(021) Ctrl memCtrl
MOV(021) &5 Ctrl
; rung 3: Descarga
LD=(300) &3 Ctrl
@AND DCarga_On  ; Descarga ativa
MOV(021) &4 Ctrl
RSET trat.FimTratamento
; rung 4: Fim Descarga
LD=(300) &4 Ctrl
ANDNOT DCarga_On  ; Descarga ativa
OUT bit_DCargaFim

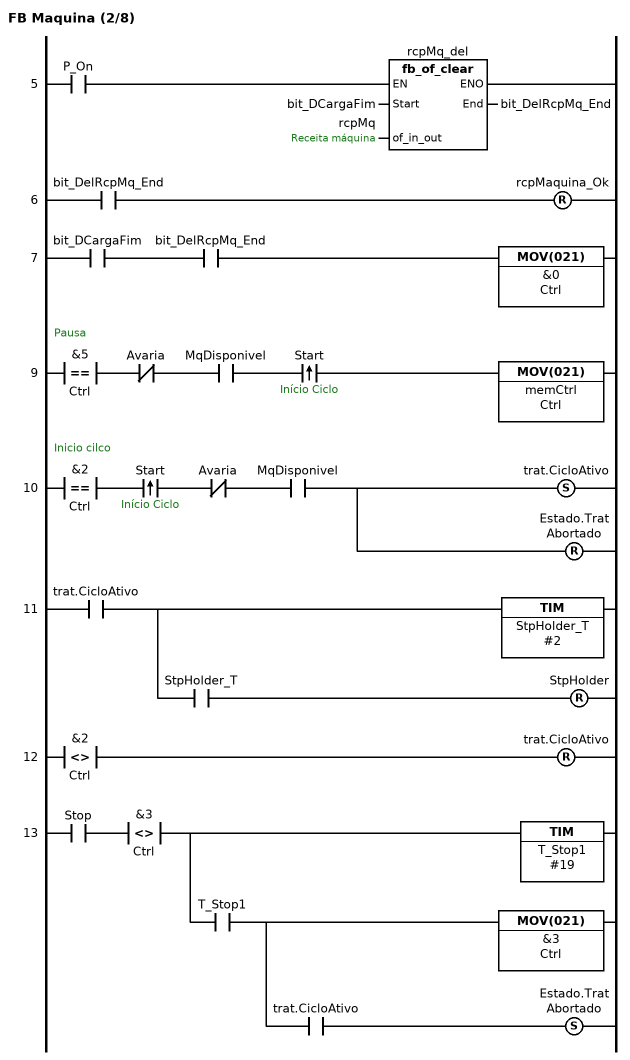
; rung 5
LD P_On
CALL rcpMq_del : fb_of_clear (Start := bit_DCargaFim, of_in_out := rcpMq, End => bit_DelRcpMq_End)  ; Receita máquina
; rung 6
LD bit_DelRcpMq_End
RSET rcpMaquina_Ok
; rung 7
LD bit_DCargaFim
AND bit_DelRcpMq_End
MOV(021) &0 Ctrl
; rung 9: Pausa
LD=(300) &5 Ctrl
ANDNOT Avaria
AND MqDisponivel
@AND Start  ; Início Ciclo
MOV(021) memCtrl Ctrl
; rung 10: Inicio cilco
LD=(300) &2 Ctrl
@AND Start  ; Início Ciclo
ANDNOT Avaria
AND MqDisponivel
SET trat.CicloAtivo
RSET Estado.TratAbortado
; rung 11
LD trat.CicloAtivo
TIM StpHolder_T #2
AND StpHolder_T
RSET StpHolder
; rung 12
LD<>(305) &2 Ctrl
RSET trat.CicloAtivo
; rung 13
LD Stop
AND<>(305) &3 Ctrl
TIM T_Stop1 #19
AND T_Stop1
MOV(021) &3 Ctrl
AND trat.CicloAtivo
SET Estado.TratAbortado

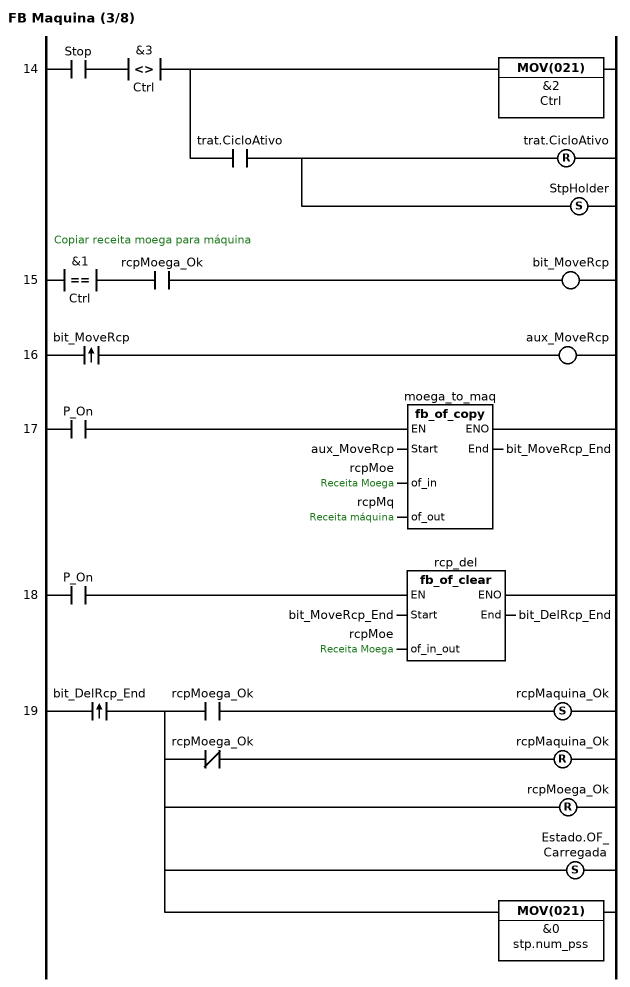
; rung 14
LD Stop
AND<>(305) &3 Ctrl
MOV(021) &2 Ctrl
AND trat.CicloAtivo
RSET trat.CicloAtivo
SET StpHolder
; rung 15: Copiar receita moega para máquina
LD=(300) &1 Ctrl
AND rcpMoega_Ok
OUT bit_MoveRcp
; rung 16
@LD bit_MoveRcp
OUT aux_MoveRcp
; rung 17
LD P_On
CALL moega_to_maq : fb_of_copy (Start := aux_MoveRcp, of_in := rcpMoe, of_out := rcpMq, End => bit_MoveRcp_End)  ; Receita Moega, Receita máquina
; rung 18
LD P_On
CALL rcp_del : fb_of_clear (Start := bit_MoveRcp_End, of_in_out := rcpMoe, End => bit_DelRcp_End)  ; Receita Moega
; rung 19
@LD bit_DelRcp_End
OUT TR0
AND rcpMoega_Ok
SET rcpMaquina_Ok
LD TR0
ANDNOT rcpMoega_Ok
RSET rcpMaquina_Ok
LD TR0
RSET rcpMoega_Ok
SET Estado.OF_Carregada
MOV(021) &0 stp.num_pss

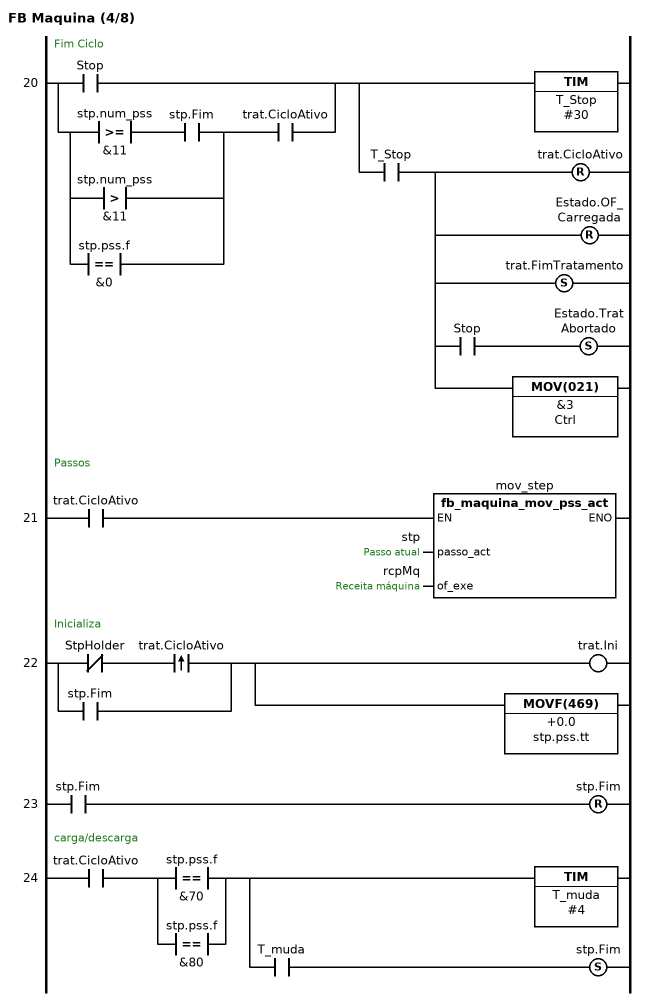
; rung 20: Fim Ciclo
LD Stop
LD>=(325) stp.num_pss &11
AND stp.Fim
OR>(320) stp.num_pss &11
OR=(300) stp.pss.f &0
AND trat.CicloAtivo
ORLD
TIM T_Stop #30
AND T_Stop
OUT TR0
RSET trat.CicloAtivo
RSET Estado.OF_Carregada
SET trat.FimTratamento
AND Stop
SET Estado.TratAbortado
LD TR0
MOV(021) &3 Ctrl
; rung 21: Passos
LD trat.CicloAtivo
CALL mov_step : fb_maquina_mov_pss_act (passo_act := stp, of_exe := rcpMq)  ; Passo atual, Receita máquina
; rung 22: Inicializa
LDNOT StpHolder
@AND trat.CicloAtivo
OR stp.Fim
OUT trat.Ini
MOVF(469) +0.0 stp.pss.tt
; rung 23
LD stp.Fim
RSET stp.Fim
; rung 24: carga/descarga
LD trat.CicloAtivo
LD=(300) stp.pss.f &70
OR=(300) stp.pss.f &80
ANDLD
TIM T_muda #4
AND T_muda
SET stp.Fim

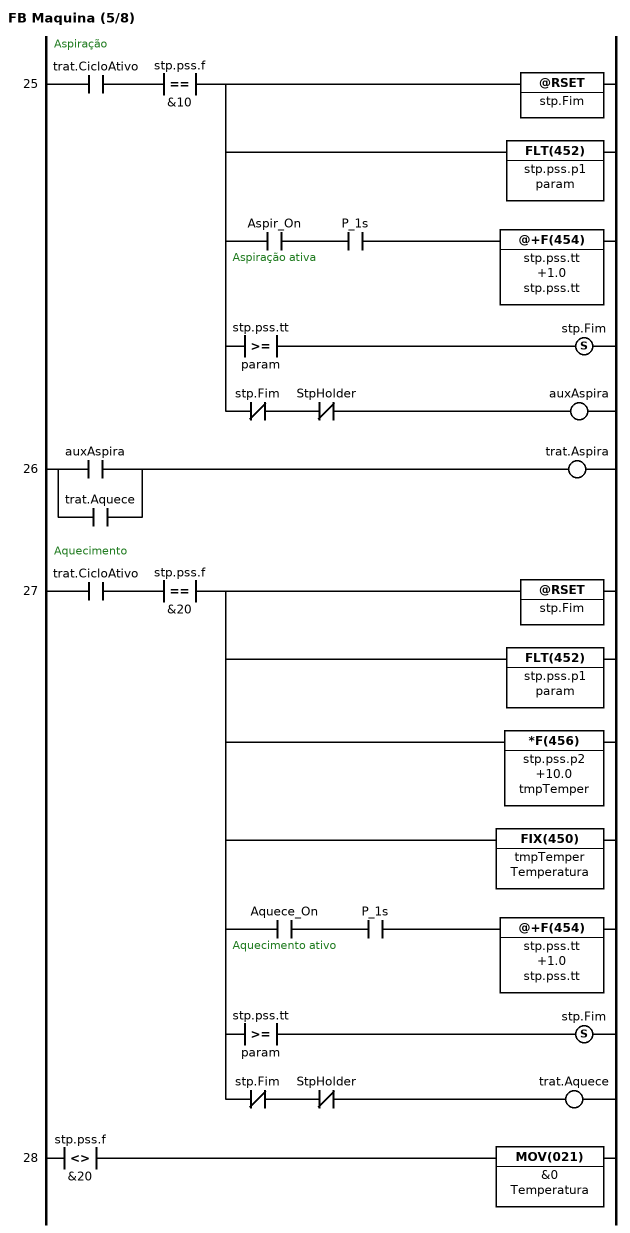
; rung 25: Aspiração
LD trat.CicloAtivo
AND=(300) stp.pss.f &10
OUT TR0
@RSET stp.Fim
FLT(452) stp.pss.p1 param
AND Aspir_On  ; Aspiração ativa
AND P_1s
@+F(454) stp.pss.tt +1.0 stp.pss.tt
LD TR0
AND>=F(334) stp.pss.tt param
SET stp.Fim
LD TR0
ANDNOT stp.Fim
ANDNOT StpHolder
OUT auxAspira
; rung 26
LD auxAspira
OR trat.Aquece
OUT trat.Aspira
; rung 27: Aquecimento
LD trat.CicloAtivo
AND=(300) stp.pss.f &20
OUT TR0
@RSET stp.Fim
FLT(452) stp.pss.p1 param
*F(456) stp.pss.p2 +10.0 tmpTemper
FIX(450) tmpTemper Temperatura
AND Aquece_On  ; Aquecimento ativo
AND P_1s
@+F(454) stp.pss.tt +1.0 stp.pss.tt
LD TR0
AND>=F(334) stp.pss.tt param
SET stp.Fim
LD TR0
ANDNOT stp.Fim
ANDNOT StpHolder
OUT trat.Aquece
; rung 28
LD<>(305) stp.pss.f &20
MOV(021) &0 Temperatura

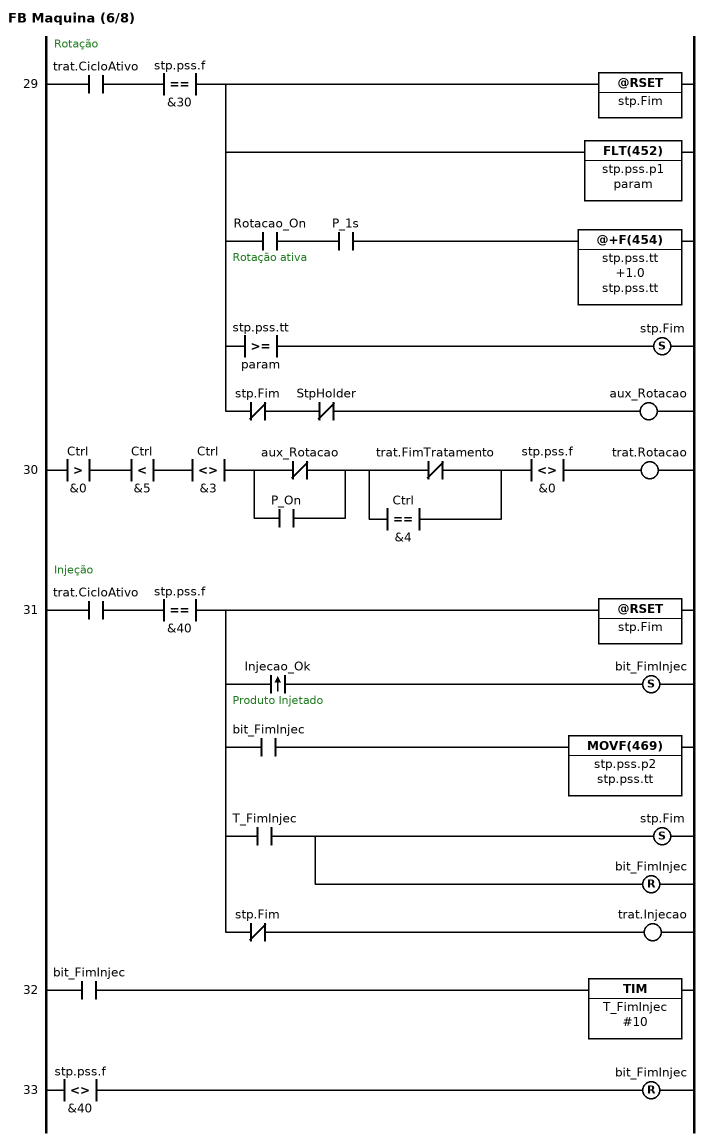
; rung 29: Rotação
LD trat.CicloAtivo
AND=(300) stp.pss.f &30
OUT TR0
@RSET stp.Fim
FLT(452) stp.pss.p1 param
AND Rotacao_On  ; Rotação ativa
AND P_1s
@+F(454) stp.pss.tt +1.0 stp.pss.tt
LD TR0
AND>=F(334) stp.pss.tt param
SET stp.Fim
LD TR0
ANDNOT stp.Fim
ANDNOT StpHolder
OUT aux_Rotacao
; rung 30
LD>(320) Ctrl &0
AND<(310) Ctrl &5
AND<>(305) Ctrl &3
LDNOT aux_Rotacao
OR P_On
ANDLD
LDNOT trat.FimTratamento
OR=(300) Ctrl &4
ANDLD
AND<>(305) stp.pss.f &0
OUT trat.Rotacao
; rung 31: Injeção
LD trat.CicloAtivo
AND=(300) stp.pss.f &40
OUT TR0
@RSET stp.Fim
@AND Injecao_Ok  ; Produto Injetado
SET bit_FimInjec
LD TR0
AND bit_FimInjec
MOVF(469) stp.pss.p2 stp.pss.tt
LD TR0
AND T_FimInjec
SET stp.Fim
RSET bit_FimInjec
LD TR0
ANDNOT stp.Fim
OUT trat.Injecao
; rung 32
LD bit_FimInjec
TIM T_FimInjec #10
; rung 33
LD<>(305) stp.pss.f &40
RSET bit_FimInjec

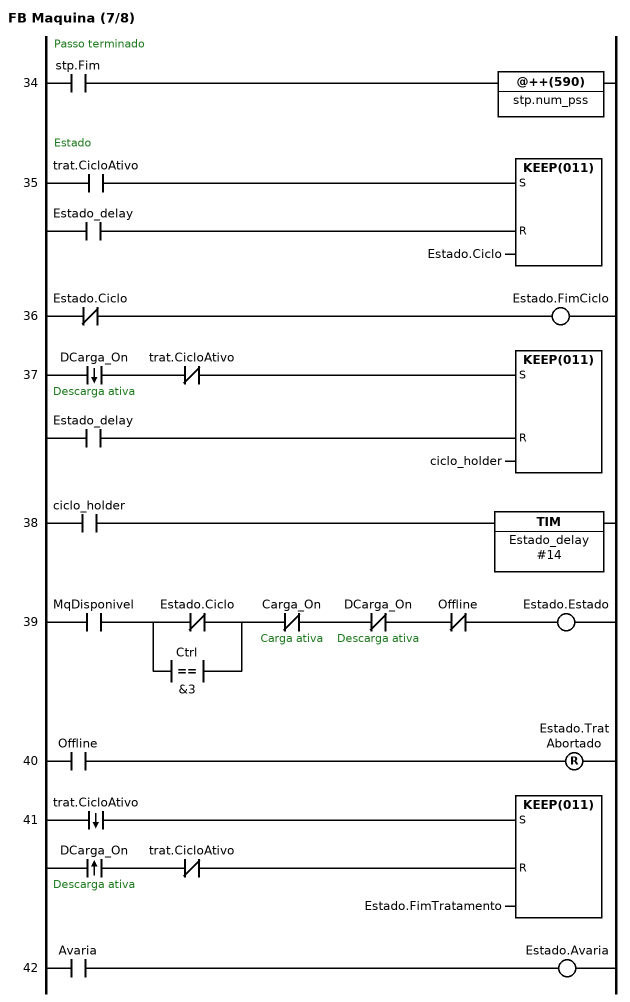
; rung 34: Passo terminado
LD stp.Fim
@++(590) stp.num_pss
; rung 35: Estado
LD trat.CicloAtivo
LD Estado_delay
KEEP(011) Estado.Ciclo
; rung 36
LDNOT Estado.Ciclo
OUT Estado.FimCiclo
; rung 37
%LD DCarga_On  ; Descarga ativa
ANDNOT trat.CicloAtivo
LD Estado_delay
KEEP(011) ciclo_holder
; rung 38
LD ciclo_holder
TIM Estado_delay #14
; rung 39
LD MqDisponivel
LDNOT Estado.Ciclo
OR=(300) Ctrl &3
ANDLD
ANDNOT Carga_On  ; Carga ativa
ANDNOT DCarga_On  ; Descarga ativa
ANDNOT Offline
OUT Estado.Estado
; rung 40
LD Offline
RSET Estado.TratAbortado
; rung 41
%LD trat.CicloAtivo
@LD DCarga_On  ; Descarga ativa
ANDNOT trat.CicloAtivo
KEEP(011) Estado.FimTratamento
; rung 42
LD Avaria
OUT Estado.Avaria

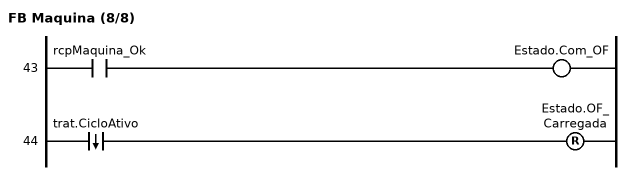
; rung 43
LD rcpMaquina_Ok
OUT Estado.Com_OF
; rung 44
%LD trat.CicloAtivo
RSET Estado.OF_Carregada